(* PLC project EPEC_CU3.project, CODESYS V3.5 SP19 *)
(* stored: creationDateTime 2026-03-19T14:01:24.6293648+02:00, modificationDateTime 2026-03-19T14:01:24.6293648+02:00 *)

(* NOTE! NOTE! NOTE! NOTE! NOTE! NOTE! NOTE! NOTE! NOTE! NOTE! NOTE! This object is created by Epec MultiTool. User changes are overwritten when project is imported. Content: - EventCode channel IDs *)
{attribute 'qualified_only'}
{attribute 'strict'}
TYPE ChannelIDs : (Ch1 := 0, Ch2, Ch3, Ch4) BYTE;
END_TYPE

(* NOTE! NOTE! NOTE! NOTE! NOTE! NOTE! NOTE! NOTE! NOTE! NOTE! NOTE! This object is created by Epec MultiTool. User changes are overwritten when project is imported. Content: - EventCode device IDs *)
{attribute 'qualified_only'}
{attribute 'strict'}
TYPE DeviceIDs : (VoltageInput := 0, DigitalInput, CurrentInput, ParameterValidation) BYTE;
END_TYPE

TYPE IdentityObject : STRUCT
  VendorId : DWORD := 0;  (* Vendor ID *)
  ProductCode : DWORD := 0;  (* Product code *)
  Revision : DWORD := 0;  (* Revision number *)
  SerialNumber : DWORD := 0;  (* Serial number for control unit *)
END_STRUCT;
END_TYPE

{attribute 'qualified_only'}
{attribute 'location' := '16#800'}
{attribute 'strict'}
TYPE InitCanProtocolStates : (INIT_CANOPEN_PROTOCOLS := 1, INIT_CANOPEN_OD := 2, INIT_CANOPEN_PDO := 3, INIT_CANOPEN_OD_SAVE := 4, INIT_CANOPEN_OD_REORG := 5, INIT_J1939 := 6, INIT_PROTOCOLS_DONE := 7);
END_TYPE

TYPE IdentityObject : STRUCT
  VendorId : DWORD := 0;  (* Vendor ID *)
  ProductCode : DWORD := 0;  (* Product code *)
  Revision : DWORD := 0;  (* Revision number *)
  SerialNumber : DWORD := 0;  (* Serial number for control unit *)
END_STRUCT;
END_TYPE

VAR_GLOBAL CONSTANT  (* G_CONSTANTS - NOTE! NOTE! NOTE! NOTE! NOTE! NOTE! NOTE! NOTE! NOTE! NOTE! NOTE! This object is created by Epec MultiTool. User changes are overwritten when project is imported. Content: - Project specific constant definitions *)
  G_PARAMHANDLERKEYWORD : DWORD := 16#30C7E7D4;  (* Parameterhandler keyword *)
  G_PARAM_BLOCK_MAX_SIZE : WORD := WORD#1024;
  G_PARAMETER_SAVE_STATUS_ERROR : BYTE := BYTE#16#00;
  G_PARAMETER_SAVE_STATUS_DONE : BYTE := BYTE#16#01;
  G_PARAMETER_SAVE_STATUS_IN_PROGRESS : BYTE := BYTE#16#FF;
  G_SAFE_PARAMETERS_AUTHENTICATED : BYTE := BYTE#1;
  G_SAFE_PARAMETERS_NOT_AUTHENTICATED : BYTE := BYTE#0;
END_VAR

{attribute 'qualified_only'}
VAR_GLOBAL  (* G_CAN - NOTE! NOTE! NOTE! NOTE! NOTE! NOTE! NOTE! NOTE! NOTE! NOTE! NOTE! This object is created by Epec MultiTool. User changes are overwritten when project is imported. Content: - CAN definitions *)
  Channel1 : EPEC_CoreCANVXD.Channel;
END_VAR

{attribute 'qualified_only'}
{attribute 'location' := '16#800'}
VAR_GLOBAL  (* G_Common *)
  ParHandler : EPEC_PH.ParameterHandler;  (* Parameterhandler. Utility library for ODSave. Library handles parameter image modification. *)
  ParFileHandler : EPEC_PH.ParameterFileHandler;  (* ParameterFileHandler. Library handles parameter image saving to file and reading it. *)
  ParameterArea : ARRAY[1..EPEC_PH.Parameters.G_PARAMETER_FILE_SIZE] OF BYTE;  (* Parameter image *)
  ProjectKey : STRING(79) := 'KEeJGzzvbvqAy4c';  (* Project key, used for validating the response code *)
END_VAR


{attribute 'qualified_only'}
{attribute 'location' := '16#800'}
{attribute 'analysis' := '-6'}
VAR_GLOBAL  (* G_Logs *)
  ApplicationLog : EPEC_SERRLOG.ErrorLog;
  AppLogInitOK : BOOL;
END_VAR


{attribute 'qualified_only'}
{attribute 'location' := '16#800'}
VAR_GLOBAL  (* G_StatusFlags - NOTE! NOTE! NOTE! NOTE! NOTE! NOTE! NOTE! NOTE! NOTE! NOTE! NOTE! This object is created by Epec MultiTool. User changes are overwritten when project is imported. Content: - PLC_PRG status flags *)
  CANopenCan1NMTResetRequest : BOOL := FALSE;  (* Reset request flags tell if module is wanted to reset after current application cycle. *)
  CANopenCan2NMTResetRequest : BOOL := FALSE;
  CANopenCan3NMTResetRequest : BOOL := FALSE;
  CANopenCan4NMTResetRequest : BOOL := FALSE;
  CANopenCan5NMTResetRequest : BOOL := FALSE;
  CANopenCan6NMTResetRequest : BOOL := FALSE;
  CANopenCan7NMTResetRequest : BOOL := FALSE;
  CANopenCan8NMTResetRequest : BOOL := FALSE;
  CANopenCan9NMTResetRequest : BOOL := FALSE;
  CANopenCan10NMTResetRequest : BOOL := FALSE;
  CANopenCan11NMTResetRequest : BOOL := FALSE;
  CANopenCan12NMTResetRequest : BOOL := FALSE;
  CANopenCan13NMTResetRequest : BOOL := FALSE;
  CANopenCan14NMTResetRequest : BOOL := FALSE;
  CANopenCan15NMTResetRequest : BOOL := FALSE;
  CANopenCan16NMTResetRequest : BOOL := FALSE;
  CANopenCan17NMTResetRequest : BOOL := FALSE;
  CANopenCan18NMTResetRequest : BOOL := FALSE;
  CANopenCan19NMTResetRequest : BOOL := FALSE;
  CANopenCan20NMTResetRequest : BOOL := FALSE;
  CANopenCan21NMTResetRequest : BOOL := FALSE;
  CANopenCan22NMTResetRequest : BOOL := FALSE;
  CANopenCan23NMTResetRequest : BOOL := FALSE;
  CANopenCan24NMTResetRequest : BOOL := FALSE;
  CANopenCan25NMTResetRequest : BOOL := FALSE;
  CANopenCan26NMTResetRequest : BOOL := FALSE;
  CANopenCan27NMTResetRequest : BOOL := FALSE;
  CANopenCan28NMTResetRequest : BOOL := FALSE;
  CANopenCan29NMTResetRequest : BOOL := FALSE;
  CANopenCan30NMTResetRequest : BOOL := FALSE;
  CANopenCan31NMTResetRequest : BOOL := FALSE;
  CANopenCan32NMTResetRequest : BOOL := FALSE;
  CANopenCan33NMTResetRequest : BOOL := FALSE;
  CANopenCan34NMTResetRequest : BOOL := FALSE;
  CANopenCan35NMTResetRequest : BOOL := FALSE;
  CANopenCan36NMTResetRequest : BOOL := FALSE;
  CANopenCan37NMTResetRequest : BOOL := FALSE;
  CANopenCan38NMTResetRequest : BOOL := FALSE;
  CANopenCan39NMTResetRequest : BOOL := FALSE;
  CANopenCan40NMTResetRequest : BOOL := FALSE;
  CANopenCan41NMTResetRequest : BOOL := FALSE;
  CANopenCan42NMTResetRequest : BOOL := FALSE;
  CANopenCan43NMTResetRequest : BOOL := FALSE;
  CANopenCan44NMTResetRequest : BOOL := FALSE;
  CANopenCan45NMTResetRequest : BOOL := FALSE;
  CANopenCan46NMTResetRequest : BOOL := FALSE;
  CANopenCan47NMTResetRequest : BOOL := FALSE;
  CANopenCan48NMTResetRequest : BOOL := FALSE;
  CANopenCan49NMTResetRequest : BOOL := FALSE;
  CANopenCan50NMTResetRequest : BOOL := FALSE;
  CANopenCan51NMTResetRequest : BOOL := FALSE;
  CANopenCan52NMTResetRequest : BOOL := FALSE;
  CANopenCan53NMTResetRequest : BOOL := FALSE;
  CANopenCan54NMTResetRequest : BOOL := FALSE;
  CANopenCan55NMTResetRequest : BOOL := FALSE;
  CANopenCan56NMTResetRequest : BOOL := FALSE;
  CANopenCan57NMTResetRequest : BOOL := FALSE;
  CANopenCan58NMTResetRequest : BOOL := FALSE;
  CANopenCan59NMTResetRequest : BOOL := FALSE;
  CANopenCan60NMTResetRequest : BOOL := FALSE;
  CANopenCan61NMTResetRequest : BOOL := FALSE;
  CANopenCan62NMTResetRequest : BOOL := FALSE;
  CANopenCan63NMTResetRequest : BOOL := FALSE;
  CANopenCan64NMTResetRequest : BOOL := FALSE;
  CANopenCan65NMTResetRequest : BOOL := FALSE;
  CANopenCan66NMTResetRequest : BOOL := FALSE;
  CANopenCan67NMTResetRequest : BOOL := FALSE;
  CANopenCan68NMTResetRequest : BOOL := FALSE;
  CANopenCan69NMTResetRequest : BOOL := FALSE;
  CANopenCan70NMTResetRequest : BOOL := FALSE;
  CANopenCan71NMTResetRequest : BOOL := FALSE;
  CANopenCan72NMTResetRequest : BOOL := FALSE;
  CANopenCan73NMTResetRequest : BOOL := FALSE;
  CANopenCan74NMTResetRequest : BOOL := FALSE;
  CANopenCan75NMTResetRequest : BOOL := FALSE;
  CANopenCan76NMTResetRequest : BOOL := FALSE;
  CANopenCan77NMTResetRequest : BOOL := FALSE;
  CANopenCan78NMTResetRequest : BOOL := FALSE;
  CANopenCan79NMTResetRequest : BOOL := FALSE;
  CANopenCan80NMTResetRequest : BOOL := FALSE;
  CANopenCan81NMTResetRequest : BOOL := FALSE;
  CANopenCan82NMTResetRequest : BOOL := FALSE;
  CANopenCan83NMTResetRequest : BOOL := FALSE;
  CANopenCan84NMTResetRequest : BOOL := FALSE;
  CANopenCan85NMTResetRequest : BOOL := FALSE;
  CANopenCan86NMTResetRequest : BOOL := FALSE;
  CANopenCan87NMTResetRequest : BOOL := FALSE;
  CANopenCan88NMTResetRequest : BOOL := FALSE;
  CANopenCan89NMTResetRequest : BOOL := FALSE;
  CANopenCan90NMTResetRequest : BOOL := FALSE;
  CANopenCan91NMTResetRequest : BOOL := FALSE;
  CANopenCan92NMTResetRequest : BOOL := FALSE;
  CANopenCan93NMTResetRequest : BOOL := FALSE;
  CANopenCan94NMTResetRequest : BOOL := FALSE;
  CANopenCan95NMTResetRequest : BOOL := FALSE;
  CANopenCan96NMTResetRequest : BOOL := FALSE;
  CANopenCan97NMTResetRequest : BOOL := FALSE;
  CANopenCan98NMTResetRequest : BOOL := FALSE;
  CANopenCan99NMTResetRequest : BOOL := FALSE;
  CANopenCan100NMTResetRequest : BOOL := FALSE;
  CANopenCan101NMTResetRequest : BOOL := FALSE;
  CANopenCan102NMTResetRequest : BOOL := FALSE;
  CANopenCan103NMTResetRequest : BOOL := FALSE;
  CANopenCan104NMTResetRequest : BOOL := FALSE;
  CANopenCan105NMTResetRequest : BOOL := FALSE;
  SystemOk : BOOL := FALSE;
END_VAR

{attribute 'qualified_only'}
{attribute 'location' := '16#800'}
VAR_GLOBAL  (* G_SystemInfo - NOTE! NOTE! NOTE! NOTE! NOTE! NOTE! NOTE! NOTE! NOTE! NOTE! NOTE! This object is created by Epec MultiTool. User changes are overwritten when project is imported. Content: - System information common for all ODs. *)
  ProjectInfo : PROJECT_INFO;
  DeviceName : STRING(79);  (* 16#1008: Manufacturer device name *)
  HWVersion : STRING(79);  (* 16#1009: Manufacturer hardware version *)
  SWVersion : STRING(79);  (* 16#100A: Manufacturer software version *)
  Identity : IdentityObject;  (* 16#1018: Identity object *)
  ToolsVersion : ARRAY[1..1] OF DWORD;  (* 16#2030 Codesys version *)
  SoftwareInformation : ARRAY[1..10] OF STRING(79) := [''];  (* 16#2130 Software information Sub1: Application version Sub2: Additional version information Sub3: Reserved for future use Sub4: Reserved for future use Sub5: Reserved for future use Sub6: Reserved for future use Sub7: Reserved for future use Sub8: Reserved for future use Sub9: Reserved for future use Sub10: Reserved for future use *)
  MACAddress : ARRAY[1..6] OF BYTE := [6(0)];  (* 16#2140 MAC address Sub1: MAC address byte 1 Sub2: MAC address byte 2 Sub3: MAC address byte 3 Sub4: MAC address byte 4 Sub5: MAC address byte 5 Sub6: MAC address byte 6 *)
  EthernetConfiguration : ARRAY[1..50] OF BYTE := [50(0)];  (* 16#2141 Ethernet configuration Sub1: Ethernet enabled/disabled Sub2: DHCP on/off Sub3: Reserved Sub4: Reserved Sub5: Reserved Sub6: Reserved Sub7: Reserved Sub8: Reserved Sub9: Reserved Sub10: Reserved Sub11: Reserved Sub12: Reserved Sub13: Reserved Sub14: Reserved Sub15: Reserved Sub16: Reserved Sub17: Reserved Sub18: Netstatus Sub19: IP address highest byte Sub20: IP address 3rd byte Sub21: IP address 2nd byte Sub22: IP address lowest byte Sub23: Gateway highest byte Sub24: Gateway 3rd byte Sub25: Gateway 2nd byte Sub26: Gateway lowest byte Sub27: Netmask highest byte Sub28: Netmask 3rd byte Sub29: Netmask 2nd byte Sub30: Netmask first byte Sub31: Reserved Sub32: Reserved Sub33: Reserved Sub34: Reserved Sub35: Reserved Sub36: Reserved Sub37: Reserved Sub38: Reserved Sub39: Reserved Sub40: Reserved Sub41: Reserved Sub42: Reserved Sub43: Reserved Sub44: Reserved Sub45: Reserved Sub46: Reserved Sub47: Reserved Sub48: Reserved Sub49: Reserved Sub50: Reserved *)
END_VAR

{attribute 'qualified_only'}
{attribute 'global_init_slot' := '49991'}
VAR_GLOBAL  (* G_CANopen_CAN1 - NOTE! NOTE! NOTE! NOTE! NOTE! NOTE! NOTE! NOTE! NOTE! NOTE! NOTE! This object is created by Epec MultiTool User changes are overwritten when project is imported Content - CANopen protocol variable definitions *)
  Device : EPEC_CANopen.Device;  (* CAN device *)
  OD : EPEC_CANopen.OD;  (* Object Dictionary data *)
  ODEntrys : ARRAY[1..67] OF EPEC_CANopen.ODEntry;
  Protocols : ARRAY[1..5] OF EPEC_CANopen.ProtocolEntry;  (* Protocol data *)
  HBCallbacks : ARRAY[1..1] OF EPEC_CANopen.CANopenHBCallback := [(i_NodeID := 3, i_Time := G_CANopen_CAN1_VAR.HBCTimes[1], i_pNext := 0)];  (* Heartbeat producer/consumer *)
  HB : EPEC_CANopen.HBData;  (* Heartbeat producer/consumer protocol data *)
  HB_Handler : EPEC_CANopen.CANopenHB;  (* Heartbeat producer/consumer protocol handler *)
  MonitoredNodes : ARRAY[1..1] OF EPEC_CANopen.SlaveData := [(pHBCallback := ADR(HBCallbacks[1]), KeepAlive := FALSE, Reset := FALSE, Mandatory := TRUE, DisableStart := FALSE, QueryWithSDO := FALSE, ConfigurationDelay := 1000, SDOQueryInterval := 0, ConfigurationTimeout := 10)];  (* NMT *)
  NMT : EPEC_CANopen.NMTData;  (* NMT protocol data *)
  NMT_Handler : EPEC_CANopen.CANopenNMT;  (* NMT protocol handler *)
  SSDO : EPEC_CANopen.SSDOData;  (* SDO server protocol data *)
  SSDO_Handler : EPEC_CANopen.CANopenSDOServer;  (* SDO server protocol handler *)
  GFC : EPEC_CANopen.GFCData;  (* GFC protocol data *)
  GFC_Handler : EPEC_CANopen.CANopenGFC;  (* GFC protocol handler *)
  CSDOS : ARRAY[1..127] OF EPEC_CANopen.CANopenCSDO := [];  (* SDO client instances *)
  AppLogDomain : EPEC_CANopen.Domain;  (* 16#2171 Application log domain *)
  SaveAll : EPEC_ODSave.SaveODSaveAll;
  DeleteAll : EPEC_ODSave.SaveODDeleteAll;
  Initialize : EPEC_ODSave.SaveODInitialize;
  SaveData : ARRAY[0..3] OF EPEC_ODSave.SaveODSubIndexDescription := [(StartIndex := 16#1000, EndIndex := 16#FFFF, GroupNum := 1), (StartIndex := 16#1000, EndIndex := 16#1FFF, GroupNum := 1), (StartIndex := 16#2000, EndIndex := 16#FFFF, GroupNum := 1), (StartIndex := 16#0, EndIndex := 16#0, GroupNum := 1)];
  SaveSubData1010h : EPEC_ODSave.SaveODSubService;
  OD_ReOrg : EPEC_CANopen.CANopenODReOrg;
END_VAR

{attribute 'qualified_only'}
{attribute 'location' := '16#800'}
{attribute 'global_init_slot' := '49990'}
VAR_GLOBAL  (* G_CANopen_CAN1_VAR - NOTE! NOTE! NOTE! NOTE! NOTE! NOTE! NOTE! NOTE! NOTE! NOTE! NOTE! This object is created by Epec MultiTool User changes are overwritten when project is imported Content - *)
  OD_Error : EPEC_CANopen.Errors := EPEC_CANopen.Errors.NotInitialized;
  ODSave_Error : EPEC_ODSave.SaveODErrors;
  Callback_Error : EPEC_CANopen.Errors := EPEC_CANopen.Errors.NotInitialized;
  ProtocolAdded : ARRAY[1..5] OF BOOL := [5(0)];
  HBCTimes : ARRAY[1..1] OF UDINT := [UDINT#400];
  HB_Error : EPEC_CANopen.Errors := EPEC_CANopen.Errors.NotInitialized;
  NMT_Error : EPEC_CANopen.Errors := EPEC_CANopen.Errors.NotInitialized;
  SSDO_Error : EPEC_CANopen.Errors := EPEC_CANopen.Errors.NotInitialized;
  GFC_Error : EPEC_CANopen.Errors := EPEC_CANopen.Errors.NotInitialized;
  GFC_Status : BYTE;  (* GFC status *)
  CSDO_Error : EPEC_CANopen.Errors := EPEC_CANopen.Errors.NotInitialized;
  OD_REORG_Error : EPEC_CANopen.Errors := EPEC_CANopen.Errors.NotInitialized;
  OdReOrgReady : BOOL := FALSE;  (* OD Reorganize operation ready *)
  SaveSigns1010 : ARRAY[0..3] OF DWORD;
  InitProtocolsCanState : InitCanProtocolStates := InitCanProtocolStates.INIT_CANOPEN_PROTOCOLS;
END_VAR

{attribute 'qualified_only'}
{attribute 'location' := '16#800'}
{attribute 'analysis' := '-5, -6, -33, -43, -48'}
VAR_GLOBAL  (* G_CAN1_VAR - NOTE! NOTE! NOTE! NOTE! NOTE! NOTE! NOTE! NOTE! NOTE! NOTE! NOTE! This object is created by Epec MultiTool User changes are overwritten when project is imported Content - CANopen OD index data *)
  DeviceType_Device1 : UDINT := 405;  (* 16#1000 Information about the device type *)
  ErrorReg_Device1 : USINT := 0;  (* 16#1001 Error information *)
  TPDO_DUMMY : BYTE := 0;  (* 16#2128 PDO Dummy Variable Index *)
  RPDO_DUMMY : BYTE := 0;  (* 16#2129 PDO Dummy Variable Index *)
  Parameter_CSV_unique_ID : UINT := 16#0000;  (* 16#2131 Parameter CSV unique ID *)
END_VAR

(* This PRG contains non safety-related code. The following attribute is autogenerated. Do not remove. *)
{attribute 'location' := '16#800'}
PROGRAM NVMemory
  VAR_INPUT
    i_Initialize : BOOL := TRUE;
  END_VAR
  VAR_OUTPUT
    o_InitReady : BOOL;
  END_VAR

            IF i_Initialize THEN
	(*Init ParameterHandler to use Filesystem *)
	G_Common.ParFileHandler.Init(
		i_pParamHandler:= ADR(G_Common.ParHandler), 
		i_pParamArea:= ADR(G_Common.ParameterArea), 
		i_ParamAreaSize:= EPEC_PH.Parameters.G_PARAMETER_FILE_SIZE, 
		i_FileName:= 'parameters.img'); 

	IF G_Common.ParFileHandler.o_Ready THEN
		G_Common.ParHandler.Init(
			i_pParamArea:= ADR(G_Common.ParameterArea),
			i_ParamAreaSize:= EPEC_PH.Parameters.G_PARAMETER_FILE_SIZE,
			i_Keyword:= G_PARAMHANDLERKEYWORD,
			i_ParameterMaxDataSize:= G_PARAM_BLOCK_MAX_SIZE);

		o_InitReady:= TRUE;
	END_IF
ELSE

	G_Common.ParFileHandler.Update(i_Enable:=TRUE);


END_IF
            
          
END_PROGRAM

(* Tool version : '8.6.9547.24640' (MultiTool build version) Xml version : '1.0.0' (MultiTool xml file version) Control Unit : 'EPEC_CU3' (Name of the unit in MultiTool) Control Unit Type : 'CORE1-01-B' (Type of the unit in MultiTool, including the functional version) CODESYS Profile : 'CODESYS V3.5 SP19' (CODESYS profile that was selected in MultiTool) Device Description Version: '3.5.19.3' (Device description version that was selected in MultiTool) Export Time : '19.03.2026 14.01.24' (Date and time when exported from MultiTool) Export Path : 'C:\Codesys RPC\apps\CodesysRPC\EPEC_CU3' (Path where MultiTool exported) Project File : 'C:\Codesys RPC\apps\CodesysRPC\CodesysRPC.mtproject' (MultiTool project file name that was used) *)
{attribute 'location' := '16#800'}
PROGRAM PLC_PRG
  VAR_OUTPUT
    o_InitDone : BOOL := FALSE;
  END_VAR

            
// Initialize application log
IF NOT G_Logs.AppLogInitOK THEN
	G_Logs.AppLogInitOK := EPEC_SERRLOG.S_InitErrorLog(i_pErrorLog:= ADR(G_Logs.ApplicationLog));
END_IF

IF NOT o_InitDone AND G_Logs.AppLogInitOK THEN

    (* Code template non-safe FB initializations *)
    IF NOT Init_Entry.o_Ready THEN
        Init_Entry();
    ELSIF NOT Init_IO.o_Ready THEN
        Init_IO();
    ELSIF NOT NVMemory.o_InitReady THEN
        NVMemory(i_Initialize:=TRUE);
	ELSIF NOT Init_CAN.o_Ready THEN
		Init_CAN();
	ELSIF NOT Init_CANopen_CAN1.o_Ready THEN
		Init_CANopen_CAN1();

    ELSE
        (* User non-safe initialization *)
        MainInit(o_MainInitReady=>o_InitDone);
    END_IF
ELSE
    (* Non-safe actions to execute before non-safe main program *)
	G_CAN.Channel1.CheckMessages();
	Handle_CANopen_CAN1();


	Handle_Diagnostic();


    (* User non-safe main program *)
    Main();

    (* Non-safe actions to execute after non-safe main program *)

    NVMemory(i_Initialize:=FALSE);

    (* Boot application if NMT reset requested *)
    //IF G_StatusFlags.CANopenCan1NMTResetRequest OR G_StatusFlags.CANopenCan2NMTResetRequest THEN
    //    EPEC_SYSTEM.BOOT_APPLICATION_KILL_RTS();
    //END_IF
END_IF



              
          
END_PROGRAM

(* NOTE! NOTE! NOTE! NOTE! NOTE! NOTE! NOTE! NOTE! NOTE! NOTE! NOTE! This object is created by Epec MultiTool User changes are overwritten when project is imported Content - Initialization of CAN channels This PRG contains non safety-related code. The following attribute is autogenerated. Do not remove. *)
{attribute 'location' := '16#800'}
{attribute 'analysis' := '-9, -38'}
PROGRAM Init_CAN
  VAR_OUTPUT
    o_Ready : BOOL := FALSE;
    o_Error : BOOL := FALSE;
    o_CAN1InitError : EPEC_CANVXD.ERROR := EPEC_CANVXD.ERROR.CHANNEL_NOT_INITIALIZED;
  END_VAR

            G_CAN.Channel1.SetLoopback(i_LoopbackEnabled:=TRUE);
o_CAN1InitError := G_CAN.Channel1.InitCAN(i_Channel := 1, i_BitRate := EPEC_CANVXD.BITRATE_250K, i_Flags := 0);

IF EPEC_CANVXD.ERROR.NO_ERROR = o_CAN1InitError THEN
	o_Error := FALSE;
ELSE
	o_Error := TRUE;

	EPEC_SERRLOG.S_AddError_DWORD(i_ErrorCode:= ApplicationErrors.CAN_INIT, i_LibraryErrorCode:= INT_TO_DINT(o_CAN1InitError), i_Info1:= 0, i_Info2:= 1);
END_IF

o_Ready := TRUE;

          
END_PROGRAM

(* NOTE! NOTE! NOTE! NOTE! NOTE! NOTE! NOTE! NOTE! NOTE! NOTE! NOTE! This object is created by Epec MultiTool User changes are overwritten when project is imported Content - Set system information common for all ODs. This PRG contains non safety-related code. The following attribute is autogenerated. Do not remove. *)
{attribute 'location' := '16#800'}
{attribute 'analysis' := '-9, -19, -26'}
PROGRAM Init_Entry
  VAR_OUTPUT
    o_Ready : BOOL;
  END_VAR

            EPEC_HW.SystemParameters.ReadData();

/// 16#1008: Manufacturer device name
G_SystemInfo.DeviceName := EPEC_HW.SystemParameters.o_DeviceName;
 /// 16#1009: Manufacturer hardware version
G_SystemInfo.HWVersion := EPEC_HW.SystemParameters.o_HardwareVersion;
/// 16#100A: Manufacturer software version
G_SystemInfo.SWVersion := EPEC_HW.SystemParameters.o_SoftwareVersion;
/// 16#1018: Identity object 
G_SystemInfo.Identity.VendorId := EPEC_HW.SystemParameters.o_VendorId;          /// Vendor ID
G_SystemInfo.Identity.ProductCode := EPEC_HW.SystemParameters.o_ProductCode;    /// Product code
G_SystemInfo.Identity.Revision := EPEC_HW.SystemParameters.o_RevisionNumber;    /// Revision number
G_SystemInfo.Identity.SerialNumber := EPEC_HW.SystemParameters.o_SerialNumber;  /// Serial number for control unit
/// 16#2030 Codesys version
G_SystemInfo.ToolsVersion[1] := DWORD#50659328;

o_Ready:= TRUE;

          
END_PROGRAM

(* NOTE! NOTE! NOTE! NOTE! NOTE! NOTE! NOTE! NOTE! NOTE! NOTE! NOTE! This object is created by Epec MultiTool User changes are overwritten when project is imported Content - Non-safe system status update This PRG contains non safety-related code. The following attribute is autogenerated. Do not remove. *)
{attribute 'location' := '16#800'}
PROGRAM Handle_Diagnostic

            (* System Ok conditions *)
G_StatusFlags.SystemOk:=
		NOT Init_CAN.o_Error AND			(* No errors in bus init *)
		NOT Init_CANopen_CAN1.o_Error;



          
END_PROGRAM

(* NOTE! NOTE! NOTE! NOTE! NOTE! NOTE! NOTE! NOTE! NOTE! NOTE! NOTE! This object is created by Epec MultiTool User changes are overwritten when project is imported Content - CANopen initialization - Includes Init_CANopen_OD1 - CANopen data update This PRG contains non safety-related code. The following attribute is autogenerated. Do not remove. *)
{attribute 'location' := '16#800'}
{attribute 'analysis' := '-9, -19, -130'}
PROGRAM Init_CANopen_CAN1
  VAR_OUTPUT
    o_Ready : BOOL := FALSE;
    o_Error : BOOL := FALSE;
  END_VAR
  VAR
    odReOrgReady : BOOL := FALSE;
  END_VAR

            CASE G_CANopen_CAN1_VAR.InitProtocolsCanState OF

InitCanProtocolStates.INIT_CANOPEN_PROTOCOLS:
	G_CANopen_CAN1.Device.itfCanChannel:=G_CAN.Channel1; (*Connect device to can channel*)
	G_CANopen_CAN1.Device.NodeID := BYTE#5;
	G_CANopen_CAN1.NMT.NmtState:=EPEC_CANopen.NMTState.BootUp; (* Set NMT status to BOOTUP *)

	(*Initialize OD's data structures*)
	G_CANopen_CAN1.OD.EntryCount:=SIZEOF(G_CANopen_CAN1.ODEntrys)/SIZEOF(G_CANopen_CAN1.ODEntrys[1]); (*Max entries of given OD(CANopenDeviceODEntrys array)*)
	G_CANopen_CAN1.OD.InOrder:=FALSE; (*OD isn't in order*)
	G_CANopen_CAN1.OD.NextFree:=0; (*OD does not have any entries yet*)
	G_CANopen_CAN1.OD.pODEntry:=ADR(G_CANopen_CAN1.ODEntrys); (*Pointer to OD array*)

	(*Define NMT protocol*)
	G_CANopen_CAN1.Protocols[1].Protocol:=EPEC_CANopen.ProtocolType.NMT;
	G_CANopen_CAN1.Protocols[1].pData:=ADR(G_CANopen_CAN1.NMT);
	G_CANopen_CAN1.Protocols[1].itfProtocol:=G_CANopen_CAN1.NMT_Handler;
	G_CANopen_CAN1.Protocols[1].pError:=ADR(G_CANopen_CAN1_VAR.NMT_Error);
	G_CANopen_CAN1_VAR.ProtocolAdded[1] := CANopenDeviceAddProtocol( (* Add to protocol stack *)
		i_pDevice:=ADR(G_CANopen_CAN1.Device),
		i_pProtocol:=ADR(G_CANopen_CAN1.Protocols[1]),
	);

	(*Initialize NMT protocol*)
	IF G_CANopen_CAN1_VAR.ProtocolAdded[1] THEN
		G_CANopen_CAN1.NMT_Handler.Init(
			i_pDevice := ADR(G_CANopen_CAN1.Device),
			i_ThisIsMaster := FALSE,
			i_StartInterval :=  1000,
			i_pMonitoredNodes := ADR(G_CANopen_CAN1.MonitoredNodes),
			i_NumberOfNodes := 1,
			i_SimultaneousSlaveConfiguration := FALSE,
			i_pOdReOrg := ADR(G_CANopen_CAN1.OD_ReOrg),
			o_Error => G_CANopen_CAN1_VAR.NMT_Error
		);
	ELSE
		G_CANopen_CAN1_VAR.NMT_Error := EPEC_CANopen.Errors.ProtocolDataMissing;
	END_IF

	(*Define OD protocol*)
	G_CANopen_CAN1.Protocols[2].Protocol:=EPEC_CANopen.ProtocolType.OD;
	G_CANopen_CAN1.Protocols[2].pData:=ADR(G_CANopen_CAN1.OD);
	G_CANopen_CAN1.Protocols[2].pError:=ADR(G_CANopen_CAN1_VAR.OD_Error);
	G_CANopen_CAN1_VAR.ProtocolAdded[2] := CANopenDeviceAddProtocol( (* Add to protocol stack *)
		i_pDevice:=ADR(G_CANopen_CAN1.Device),
		i_pProtocol:=ADR(G_CANopen_CAN1.Protocols[2]),
	);
	IF NOT G_CANopen_CAN1_VAR.ProtocolAdded[2] THEN
		G_CANopen_CAN1_VAR.OD_Error := EPEC_CANopen.Errors.ProtocolDataMissing;
	END_IF

	(*Define HB protocol
	- Uses NMT and OD protocol data, thus need to be defined after them.
	*)
	G_CANopen_CAN1.HB.HeartBeat.PT := T#200MS; (* HB producer time *)
	G_CANopen_CAN1.HB.pHBCTimes := ADR(G_CANopen_CAN1_VAR.HBCTimes); (* HB consumer times *)

	G_CANopen_CAN1.Protocols[3].Protocol:=EPEC_CANopen.ProtocolType.HB;
	G_CANopen_CAN1.Protocols[3].pData:=ADR(G_CANopen_CAN1.HB);
	G_CANopen_CAN1.Protocols[3].itfProtocol:=G_CANopen_CAN1.HB_Handler;
	G_CANopen_CAN1.Protocols[3].pError:=ADR(G_CANopen_CAN1_VAR.HB_Error);
	G_CANopen_CAN1_VAR.ProtocolAdded[3] := CANopenDeviceAddProtocol( (* Add to protocol stack *)
		i_pDevice:=ADR(G_CANopen_CAN1.Device),
		i_pProtocol:=ADR(G_CANopen_CAN1.Protocols[3]),
	);

	(* Initialize HB protocol *)
	IF G_CANopen_CAN1_VAR.ProtocolAdded[3] THEN

		(* Add monitored nodes *)
		G_CANopen_CAN1.HB_Handler.AddCallbackToList(
			i_pDevice := ADR(G_CANopen_CAN1.Device),
			i_pCallback:=ADR(G_CANopen_CAN1.HBCallbacks[1]),
			o_Error => G_CANopen_CAN1_VAR.HB_Error
		);
		IF G_CANopen_CAN1_VAR.HB_Error = EPEC_CANopen.Errors.NoError THEN
			G_CANopen_CAN1.HB_Handler.Init(
				i_pDevice := ADR(G_CANopen_CAN1.Device),
				o_Error => G_CANopen_CAN1_VAR.HB_Error
			);
		END_IF
	ELSE
		G_CANopen_CAN1_VAR.HB_Error := EPEC_CANopen.Errors.ProtocolDataMissing;
	END_IF

	(*Define SSDO protocol*)
	G_CANopen_CAN1.Protocols[4].Protocol:=EPEC_CANopen.ProtocolType.SSDO;
	G_CANopen_CAN1.Protocols[4].pData:=ADR(G_CANopen_CAN1.SSDO);
	G_CANopen_CAN1.Protocols[4].itfProtocol:=G_CANopen_CAN1.SSDO_Handler;
	G_CANopen_CAN1.Protocols[4].pError:=ADR(G_CANopen_CAN1_VAR.SSDO_Error);
	G_CANopen_CAN1_VAR.ProtocolAdded[4] := CANopenDeviceAddProtocol( (* Add to protocol stack *)
		i_pDevice:=ADR(G_CANopen_CAN1.Device),
		i_pProtocol:=ADR(G_CANopen_CAN1.Protocols[4])
	);
	IF G_CANopen_CAN1_VAR.ProtocolAdded[4] THEN
		G_CANopen_CAN1.SSDO_Handler.Init(
			i_pDevice := ADR(G_CANopen_CAN1.Device),
			o_Error => G_CANopen_CAN1_VAR.SSDO_Error
		);
	ELSE
		G_CANopen_CAN1_VAR.SSDO_Error := EPEC_CANopen.Errors.ProtocolDataMissing;
	END_IF

	(*Define GFC protocol*)
	G_CANopen_CAN1.Protocols[5].Protocol:=EPEC_CANopen.ProtocolType.GFC;
	G_CANopen_CAN1.Protocols[5].pData:=ADR(G_CANopen_CAN1.GFC);
	G_CANopen_CAN1.Protocols[5].itfProtocol:=G_CANopen_CAN1.GFC_Handler;
	G_CANopen_CAN1.Protocols[5].pError:=ADR(G_CANopen_CAN1_VAR.GFC_Error);
	G_CANopen_CAN1_VAR.ProtocolAdded[5] := CANopenDeviceAddProtocol(  (* Add to protocol stack *)
		i_pDevice:=ADR(G_CANopen_CAN1.Device),
		i_pProtocol:=ADR(G_CANopen_CAN1.Protocols[5])
	);
	IF G_CANopen_CAN1_VAR.ProtocolAdded[5] THEN
		G_CANopen_CAN1.GFC_Handler.Init(
			i_pDevice := ADR(G_CANopen_CAN1.Device),
			i_pStatus:=ADR(G_CANopen_CAN1_VAR.GFC_Status),
			o_Error => G_CANopen_CAN1_VAR.GFC_Error
		);
	ELSE
		G_CANopen_CAN1_VAR.GFC_Error := EPEC_CANopen.Errors.ProtocolDataMissing;
	END_IF

	(* Init CSDO instance array for bus *)
	EPEC_CANopen.CANopenSDOManager.Init(
		i_pDevice:=ADR(G_CANopen_CAN1.Device),
		i_pCSDOArrayStart:=ADR(G_CANopen_CAN1.CSDOS),
		i_CSDOArraySize:=SIZEOF(G_CANopen_CAN1.CSDOS)/SIZEOF(G_CANopen_CAN1.CSDOS[1]),
		o_Error=>G_CANopen_CAN1_VAR.CSDO_Error
	);

	G_CANopen_CAN1_VAR.InitProtocolsCanState := InitCanProtocolStates.INIT_CANOPEN_OD;

InitCanProtocolStates.INIT_CANOPEN_OD:

	(* Add index data to OD *)
	Init_CANopen_OD1(o_Ready=>); (* Must be done before initing PDOs and SRDOs. *)

	IF Init_CANopen_OD1.o_Ready THEN
		G_CANopen_CAN1_VAR.InitProtocolsCanState := InitCanProtocolStates.INIT_CANOPEN_OD_SAVE;
	END_IF


InitCanProtocolStates.INIT_CANOPEN_OD_SAVE:

	(*Initialize OD save*)
	G_CANopen_CAN1.SaveAll.Init(i_pParamHandler:=ADR(G_Common.ParHandler));
	G_CANopen_CAN1.DeleteAll.Init(i_pParamHandler:=ADR(G_Common.ParHandler));
	G_CANopen_CAN1.SaveSubData1010h.pSaveSigns := ADR(G_CANopen_CAN1_VAR.SaveSigns1010[0]);
	G_CANopen_CAN1.SaveSubData1010h.NumOfEntrys := 4;
	G_CANopen_CAN1.SaveSubData1010h.pSaveIndexData := ADR(G_CANopen_CAN1.SaveData[0]);
	G_CANopen_CAN1.SaveData[3].itfSaveAll := G_CANopen_CAN1.SaveAll;
	G_CANopen_CAN1.SaveData[3].itfDeleteAll := G_CANopen_CAN1.DeleteAll;
	G_CANopen_CAN1.OD.pAdditionalData := ADR(G_CANopen_CAN1.SaveSubData1010h);

	IF G_CANopen_CAN1_VAR.OD_Error = EPEC_CANopen.Errors.NoError THEN
		G_CANopen_CAN1.Initialize(i_pOD:=ADR(G_CANopen_CAN1.OD), i_pParamHandler:=ADR(G_Common.ParHandler), o_Error => G_CANopen_CAN1_VAR.ODSave_Error);
	END_IF

	G_CANopen_CAN1.OD_ReOrg.Init(i_pOD := ADR(G_CANopen_CAN1.OD), i_NumOfODIndexPerCycle := 50);
	G_CANopen_CAN1.OD_ReOrg.Start();

	G_CANopen_CAN1_VAR.InitProtocolsCanState := InitCanProtocolStates.INIT_CANOPEN_OD_REORG;

InitCanProtocolStates.INIT_CANOPEN_OD_REORG:

	G_CANopen_CAN1.OD_ReOrg.Update(o_Ready => odReOrgReady, o_Error => G_CANopen_CAN1_VAR.OD_REORG_Error);

	IF odReOrgReady THEN
		(* Check all protocol init status flags *)
		IF G_CANopen_CAN1_VAR.NMT_Error = EPEC_CANopen.Errors.NoError AND
			G_CANopen_CAN1_VAR.SSDO_Error = EPEC_CANopen.Errors.NoError AND
			G_CANopen_CAN1_VAR.OD_Error = EPEC_CANopen.Errors.NoError AND
			G_CANopen_CAN1_VAR.HB_Error = EPEC_CANopen.Errors.NoError AND
			G_CANopen_CAN1_VAR.CSDO_Error = EPEC_CANopen.Errors.NoError AND
			G_CANopen_CAN1_VAR.GFC_Error = EPEC_CANopen.Errors.NoError AND
			G_CANopen_CAN1_VAR.OD_REORG_Error = EPEC_CANopen.Errors.NoError
		THEN
			o_Error := FALSE; (* No errors in protocol inits *)
		ELSE
			o_Error := TRUE;

			EPEC_SERRLOG.S_AddError_DWORD(i_ErrorCode:= ApplicationErrors.CANOPEN_INIT_NMT, i_LibraryErrorCode:= INT_TO_DINT(G_CANopen_CAN1_VAR.NMT_Error), i_Info1:= 0, i_Info2:= 1);
			EPEC_SERRLOG.S_AddError_DWORD(i_ErrorCode:= ApplicationErrors.CANOPEN_INIT_SSDO, i_LibraryErrorCode:= INT_TO_DINT(G_CANopen_CAN1_VAR.SSDO_Error), i_Info1:= 0, i_Info2:= 1);
			EPEC_SERRLOG.S_AddError_DWORD(i_ErrorCode:= ApplicationErrors.CANOPEN_INIT_OD, i_LibraryErrorCode:= INT_TO_DINT(G_CANopen_CAN1_VAR.OD_Error), i_Info1:= 0, i_Info2:= 1);
			EPEC_SERRLOG.S_AddError_DWORD(i_ErrorCode:= ApplicationErrors.CANOPEN_INIT_HB, i_LibraryErrorCode:= INT_TO_DINT(G_CANopen_CAN1_VAR.HB_Error), i_Info1:= 0, i_Info2:= 1);
			EPEC_SERRLOG.S_AddError_DWORD(i_ErrorCode:= ApplicationErrors.CANOPEN_INIT_CSDO, i_LibraryErrorCode:= INT_TO_DINT(G_CANopen_CAN1_VAR.CSDO_Error), i_Info1:= 0, i_Info2:= 1);
			EPEC_SERRLOG.S_AddError_DWORD(i_ErrorCode:= ApplicationErrors.CANOPEN_INIT_GFC, i_LibraryErrorCode:= INT_TO_DINT(G_CANopen_CAN1_VAR.GFC_Error), i_Info1:= 0, i_Info2:= 1);
			EPEC_SERRLOG.S_AddError_DWORD(i_ErrorCode:= ApplicationErrors.CANOPEN_INIT_OD_REORG, i_LibraryErrorCode:= INT_TO_DINT(G_CANopen_CAN1_VAR.OD_REORG_Error), i_Info1:= 0, i_Info2:= 1);

		END_IF

		o_Ready:=TRUE;
		G_CANopen_CAN1_VAR.InitProtocolsCanState := InitCanProtocolStates.INIT_PROTOCOLS_DONE;
	END_IF
END_CASE

          
END_PROGRAM

(* NOTE! NOTE! NOTE! NOTE! NOTE! NOTE! NOTE! NOTE! NOTE! NOTE! NOTE! This object is created by Epec MultiTool User changes are overwritten when project is imported Content - CANopen object dictionary initialization This PRG contains non safety-related code. The following attribute is autogenerated. Do not remove. *)
{attribute 'location' := '16#800'}
{attribute 'analysis' := '-19'}
PROGRAM Init_CANopen_OD1
  VAR_OUTPUT
    o_Ready : BOOL := FALSE;
  END_VAR

            CASE G_CANopen_CAN1_VAR.InitProtocolsCanState OF

InitCanProtocolStates.INIT_CANOPEN_OD:

	(*16#0001..16#0009 Default types *)
	G_CANopen_CAN1_VAR.OD_Error := EPEC_CANopen.CANopenODAddDefautTypes(
		i_pOD:= ADR(G_CANopen_CAN1.OD)
	);

	(* 16#1000 Information about the device type *)
	IF G_CANopen_CAN1_VAR.OD_Error = EPEC_CANopen.Errors.NoError THEN
		G_CANopen_CAN1_VAR.OD_Error := CANopenODAddLine(
			i_pOD := ADR(G_CANopen_CAN1.OD),(*Address of Object dictionary where index will be added*)
			i_Index := G_CANOPEN_ODINDEX_DEVICE_TYPE,
			i_ObjectCode := EPEC_CANopen.ObjectCode.OD_VAR,(*Type of index*)
			i_NumOfSubids := USINT#0,(*Number of subindexes*)
			i_TypeSpec := EPEC_CANopen.DataType.Deftype_UNSIGNED32,(*Index datatype, either user defined or standard CiA 301*)
			i_ObjectAccess := G_CANOPEN_OD_ACCESS_NOWRITE OR G_CANOPEN_OD_ACCESS_SUB0NOWRITE,
			i_Sub0data := USINT#0,(*Value of subindex0 in array or (def)struct*)
			i_pIndexData := ADR(G_CAN1_VAR.DeviceType_Device1),
			i_itfSDOHandler := DWORD#0
		);
	END_IF

	(* 16#1001 Error information *)
	IF G_CANopen_CAN1_VAR.OD_Error = EPEC_CANopen.Errors.NoError THEN
		G_CANopen_CAN1_VAR.OD_Error := CANopenODAddLine(
			i_pOD := ADR(G_CANopen_CAN1.OD),(*Address of Object dictionary where index will be added*)
			i_Index := G_CANOPEN_ODINDEX_ERROR_REGISTER,
			i_ObjectCode := EPEC_CANopen.ObjectCode.OD_VAR,(*Type of index*)
			i_NumOfSubids := USINT#0,(*Number of subindexes*)
			i_TypeSpec := EPEC_CANopen.DataType.Deftype_UNSIGNED8,(*Index datatype, either user defined or standard CiA 301*)
			i_ObjectAccess := G_CANOPEN_OD_ACCESS_NOWRITE OR G_CANOPEN_OD_ACCESS_SUB0NOWRITE,
			i_Sub0data := USINT#0,(*Value of subindex0 in array or (def)struct*)
			i_pIndexData := ADR(G_CAN1_VAR.ErrorReg_Device1),
			i_itfSDOHandler := DWORD#0
		);
	END_IF

	(* 16#1008 Manufacturer device name *)
	IF G_CANopen_CAN1_VAR.OD_Error = EPEC_CANopen.Errors.NoError THEN
		G_CANopen_CAN1_VAR.OD_Error := CANopenODAddLine(
			i_pOD := ADR(G_CANopen_CAN1.OD),(*Address of Object dictionary where index will be added*)
			i_Index := G_CANOPEN_ODINDEX_MF_DEVICE_NAME,
			i_ObjectCode := EPEC_CANopen.ObjectCode.OD_VAR,(*Type of index*)
			i_NumOfSubids := USINT#0,(*Number of subindexes*)
			i_TypeSpec := EPEC_CANopen.DataType.Deftype_STRING,(*Index datatype, either user defined or standard CiA 301*)
			i_ObjectAccess := G_CANOPEN_OD_ACCESS_NOWRITE OR G_CANOPEN_OD_ACCESS_SUB0NOWRITE,
			i_Sub0data := USINT#0,(*Value of subindex0 in array or (def)struct*)
			i_pIndexData := ADR(G_SystemInfo.DeviceName),
			i_itfSDOHandler := DWORD#0
		);
	END_IF

	(* 16#100A Manufacturer software version *)
	IF G_CANopen_CAN1_VAR.OD_Error = EPEC_CANopen.Errors.NoError THEN
		G_CANopen_CAN1_VAR.OD_Error := CANopenODAddLine(
			i_pOD := ADR(G_CANopen_CAN1.OD),(*Address of Object dictionary where index will be added*)
			i_Index := G_CANOPEN_ODINDEX_MF_SW_VERSION,
			i_ObjectCode := EPEC_CANopen.ObjectCode.OD_VAR,(*Type of index*)
			i_NumOfSubids := USINT#0,(*Number of subindexes*)
			i_TypeSpec := EPEC_CANopen.DataType.Deftype_STRING,(*Index datatype, either user defined or standard CiA 301*)
			i_ObjectAccess := G_CANOPEN_OD_ACCESS_NOWRITE OR G_CANOPEN_OD_ACCESS_SUB0NOWRITE,
			i_Sub0data := USINT#0,(*Value of subindex0 in array or (def)struct*)
			i_pIndexData := ADR(G_SystemInfo.SWVersion),
			i_itfSDOHandler := DWORD#0
		);
	END_IF

	(* 16#1018   Vendor ID *)
	IF G_CANopen_CAN1_VAR.OD_Error = EPEC_CANopen.Errors.NoError THEN
		G_CANopen_CAN1_VAR.OD_Error := CANopenODAddLine(
			i_pOD := ADR(G_CANopen_CAN1.OD),(*Address of Object dictionary where index will be added*)
			i_Index := G_CANOPEN_ODINDEX_IDENTITY_OBJECT,
			i_ObjectCode := EPEC_CANopen.ObjectCode.OD_ARRAY, (*Type of index*)
			i_NumOfSubids := USINT#4,(*Number of subindexes*)
			i_TypeSpec := EPEC_CANopen.DataType.Deftype_UNSIGNED32,(*Index of 16-bit deftype*)
			i_ObjectAccess := G_CANOPEN_OD_ACCESS_NOWRITE OR G_CANOPEN_OD_ACCESS_SUB0NOWRITE,
			i_Sub0data := USINT#4,(*Value of subindex0 in array or (def)struct*)
			i_pIndexData := ADR(G_SystemInfo.Identity),
			i_itfSDOHandler := DWORD#0
		);
	END_IF
	(* 16#2030   CodesysVersion *)
	IF G_CANopen_CAN1_VAR.OD_Error = EPEC_CANopen.Errors.NoError THEN
		G_CANopen_CAN1_VAR.OD_Error := CANopenODAddLine(
			i_pOD := ADR(G_CANopen_CAN1.OD),(*Address of Object dictionary where index will be added*)
			i_Index := 16#2030,
			i_ObjectCode := EPEC_CANopen.ObjectCode.OD_ARRAY, (*Type of index*)
			i_NumOfSubids := USINT#1,(*Number of subindexes*)
			i_TypeSpec := EPEC_CANopen.DataType.Deftype_UNSIGNED32,(*Index of 16-bit deftype*)
			i_ObjectAccess := G_CANOPEN_OD_ACCESS_NOWRITE OR G_CANOPEN_OD_ACCESS_SUB0NOWRITE,
			i_Sub0data := USINT#1,(*Value of subindex0 in array or (def)struct*)
			i_pIndexData := ADR(G_SystemInfo.ToolsVersion),
			i_itfSDOHandler := DWORD#0
		);
	END_IF

	(* 16#2128 PDO Dummy Variable Index *)
	IF G_CANopen_CAN1_VAR.OD_Error = EPEC_CANopen.Errors.NoError THEN
		G_CANopen_CAN1_VAR.OD_Error := CANopenODAddLine(
			i_pOD := ADR(G_CANopen_CAN1.OD),(*Address of Object dictionary where index will be added*)
			i_Index := 16#2128,
			i_ObjectCode := EPEC_CANopen.ObjectCode.OD_VAR,(*Type of index*)
			i_NumOfSubids := USINT#0,(*Number of subindexes*)
			i_TypeSpec := EPEC_CANopen.DataType.Deftype_UNSIGNED8,(*Index datatype, either user defined or standard CiA 301*)
			i_ObjectAccess := G_CANOPEN_OD_ACCESS_READWRITE,
			i_Sub0data := USINT#0,(*Value of subindex0 in array or (def)struct*)
			i_pIndexData := ADR(G_CAN1_VAR.TPDO_DUMMY),
			i_itfSDOHandler := DWORD#0
		);
	END_IF

	(* 16#2129 PDO Dummy Variable Index *)
	IF G_CANopen_CAN1_VAR.OD_Error = EPEC_CANopen.Errors.NoError THEN
		G_CANopen_CAN1_VAR.OD_Error := CANopenODAddLine(
			i_pOD := ADR(G_CANopen_CAN1.OD),(*Address of Object dictionary where index will be added*)
			i_Index := 16#2129,
			i_ObjectCode := EPEC_CANopen.ObjectCode.OD_VAR,(*Type of index*)
			i_NumOfSubids := USINT#0,(*Number of subindexes*)
			i_TypeSpec := EPEC_CANopen.DataType.Deftype_UNSIGNED8,(*Index datatype, either user defined or standard CiA 301*)
			i_ObjectAccess := G_CANOPEN_OD_ACCESS_READWRITE,
			i_Sub0data := USINT#0,(*Value of subindex0 in array or (def)struct*)
			i_pIndexData := ADR(G_CAN1_VAR.RPDO_DUMMY),
			i_itfSDOHandler := DWORD#0
		);
	END_IF

	(* 16#2130   Application version *)
	IF G_CANopen_CAN1_VAR.OD_Error = EPEC_CANopen.Errors.NoError THEN
		G_CANopen_CAN1_VAR.OD_Error := CANopenODAddLine(
			i_pOD := ADR(G_CANopen_CAN1.OD),(*Address of Object dictionary where index will be added*)
			i_Index := 16#2130,
			i_ObjectCode := EPEC_CANopen.ObjectCode.OD_ARRAY, (*Type of index*)
			i_NumOfSubids := USINT#10,(*Number of subindexes*)
			i_TypeSpec := EPEC_CANopen.DataType.Deftype_STRING,(*Index of 16-bit deftype*)
			i_ObjectAccess := G_CANOPEN_OD_ACCESS_NOWRITE OR G_CANOPEN_OD_ACCESS_SUB0NOWRITE,
			i_Sub0data := USINT#10,(*Value of subindex0 in array or (def)struct*)
			i_pIndexData := ADR(G_SystemInfo.SoftwareInformation),
			i_itfSDOHandler := DWORD#0
		);
	END_IF

	(* 16#2140   MAC address byte 1 *)
	IF G_CANopen_CAN1_VAR.OD_Error = EPEC_CANopen.Errors.NoError THEN
		G_CANopen_CAN1_VAR.OD_Error := CANopenODAddLine(
			i_pOD := ADR(G_CANopen_CAN1.OD),(*Address of Object dictionary where index will be added*)
			i_Index := 16#2140,
			i_ObjectCode := EPEC_CANopen.ObjectCode.OD_ARRAY, (*Type of index*)
			i_NumOfSubids := USINT#6,(*Number of subindexes*)
			i_TypeSpec := EPEC_CANopen.DataType.Deftype_UNSIGNED8,(*Index of 16-bit deftype*)
			i_ObjectAccess := G_CANOPEN_OD_ACCESS_NOWRITE OR G_CANOPEN_OD_ACCESS_SUB0NOWRITE,
			i_Sub0data := USINT#6,(*Value of subindex0 in array or (def)struct*)
			i_pIndexData := ADR(G_SystemInfo.MACAddress),
			i_itfSDOHandler := DWORD#0
		);
	END_IF

	(* 16#2141   Ethernet enabled/disabled *)
	IF G_CANopen_CAN1_VAR.OD_Error = EPEC_CANopen.Errors.NoError THEN
		G_CANopen_CAN1_VAR.OD_Error := CANopenODAddLine(
			i_pOD := ADR(G_CANopen_CAN1.OD),(*Address of Object dictionary where index will be added*)
			i_Index := 16#2141,
			i_ObjectCode := EPEC_CANopen.ObjectCode.OD_ARRAY, (*Type of index*)
			i_NumOfSubids := USINT#50,(*Number of subindexes*)
			i_TypeSpec := EPEC_CANopen.DataType.Deftype_UNSIGNED8,(*Index of 16-bit deftype*)
			i_ObjectAccess := G_CANOPEN_OD_ACCESS_READWRITE OR G_CANOPEN_OD_ACCESS_SUB0NOWRITE,
			i_Sub0data := USINT#50,(*Value of subindex0 in array or (def)struct*)
			i_pIndexData := ADR(G_SystemInfo.EthernetConfiguration),
			i_itfSDOHandler := DWORD#0
		);
	END_IF

	(* 16#2131 Parameter CSV unique ID *)
	IF G_CANopen_CAN1_VAR.OD_Error = EPEC_CANopen.Errors.NoError THEN
		G_CANopen_CAN1_VAR.OD_Error := CANopenODAddLine(
			i_pOD := ADR(G_CANopen_CAN1.OD),(*Address of Object dictionary where index will be added*)
			i_Index := 16#2131,
			i_ObjectCode := EPEC_CANopen.ObjectCode.OD_VAR,(*Type of index*)
			i_NumOfSubids := USINT#0,(*Number of subindexes*)
			i_TypeSpec := EPEC_CANopen.DataType.Deftype_UNSIGNED16,(*Index datatype, either user defined or standard CiA 301*)
			i_ObjectAccess := G_CANOPEN_OD_ACCESS_NOWRITE OR G_CANOPEN_OD_ACCESS_SUB0NOWRITE,
			i_Sub0data := USINT#0,(*Value of subindex0 in array or (def)struct*)
			i_pIndexData := ADR(G_CAN1_VAR.Parameter_CSV_unique_ID),
			i_itfSDOHandler := DWORD#0
		);
	END_IF

	(*16#2170 Application log error count *)
	IF G_CANopen_CAN1_VAR.OD_Error = EPEC_CANopen.Errors.NoError THEN
		G_CANopen_CAN1_VAR.OD_Error := CANopenODAddLine(
			i_pOD:= ADR(G_CANopen_CAN1.OD), (*Address of Object dictionary where index will be added *)
			i_Index:= 16#2170,
			i_ObjectCode:= EPEC_CANopen.ObjectCode.OD_VAR, (*Type of index*)
			i_NumOfSubids:= USINT#0,(*Number of subindexes*)
			i_TypeSpec:= EPEC_CANopen.DataType.Deftype_UNSIGNED32,(*Index of 32 - bit deftype *)
			i_ObjectAccess:= G_CANOPEN_OD_ACCESS_NOWRITE OR G_CANOPEN_OD_ACCESS_SUB0NOWRITE,
			i_Sub0data := USINT#0,(*Value of subindex0 in array or (def)struct*)
			i_pIndexData:= ADR(G_Logs.ApplicationLog.count),
			i_itfSDOHandler:= DWORD#0
		);
	END_IF

	(*16#2171 Application log domain *)
		IF G_CANopen_CAN1_VAR.OD_Error = EPEC_CANopen.Errors.NoError THEN
		G_CANopen_CAN1.AppLogDomain.DataSize:= SIZEOF(G_Logs.ApplicationLog.loglines) * 8;
		G_CANopen_CAN1.AppLogDomain.pData:= ADR(G_Logs.ApplicationLog.loglines);

		G_CANopen_CAN1_VAR.OD_Error := CANopenODAddLine(
			i_pOD:= ADR(G_CANopen_CAN1.OD), (*Address of Object dictionary where index will be added *)
			i_Index:= 16#2171,
			i_ObjectCode:= EPEC_CANopen.ObjectCode.OD_DOMAIN, (*Type of index*)
			i_NumOfSubids:= USINT#0,(*Number of subindexes*)
			i_TypeSpec:= EPEC_CANopen.DataType.Deftype_Domain,(*Domain deftype *)
			i_ObjectAccess:= G_CANOPEN_OD_ACCESS_NOWRITE,
			i_Sub0data:= USINT#0,(*Value of subindex0 in array or (def)struct*)
			i_pIndexData:= ADR(G_CANopen_CAN1.AppLogDomain),
			i_itfSDOHandler:= DWORD#0
		);
	END_IF

	o_Ready := TRUE;
END_CASE

          
END_PROGRAM

(* NOTE! NOTE! NOTE! NOTE! NOTE! NOTE! NOTE! NOTE! NOTE! NOTE! NOTE! This object is created by Epec MultiTool User changes are overwritten when project is imported Content - CANopen data update This PRG contains non safety-related code. The following attribute is autogenerated. Do not remove. *)
{attribute 'location' := '16#800'}
{attribute 'analysis' := '-9, -169'}
PROGRAM Handle_CANopen_CAN1
  VAR_OUTPUT
    o_Error : BOOL := FALSE;
  END_VAR

            (* Update callback data *)
IF G_CAN.Channel1.GetLatestError() <> DWORD#0 THEN
	G_CANopen_CAN1_VAR.Callback_Error := EPEC_CANopen.Errors.CallbackError;
ELSE
	G_CANopen_CAN1_VAR.Callback_Error := EPEC_CANopen.Errors.NoError;
END_IF

(* Update protocol data *)
G_CANopen_CAN1.HB_Handler.Update(
	i_Enable := TRUE,
	o_Error => G_CANopen_CAN1_VAR.HB_Error
);
G_CANopen_CAN1.NMT_Handler.Update(
	i_Enable := TRUE,
	o_Error => G_CANopen_CAN1_VAR.NMT_Error
);
G_CANopen_CAN1.SSDO_Handler.Update(
	i_Enable := TRUE,
	o_Error => G_CANopen_CAN1_VAR.SSDO_Error
);
G_CANopen_CAN1.GFC_Handler.Update(
	i_Enable := TRUE,
	o_Error => G_CANopen_CAN1_VAR.GFC_Error
);

G_CANopen_CAN1.OD_ReOrg.Update(o_Ready => , o_Error => G_CANopen_CAN1_VAR.OD_REORG_Error);

IF G_CANopen_CAN1_VAR.HB_Error = EPEC_CANopen.Errors.NoError AND
	G_CANopen_CAN1_VAR.NMT_Error = EPEC_CANopen.Errors.NoError AND
	G_CANopen_CAN1_VAR.SSDO_Error = EPEC_CANopen.Errors.NoError AND
	G_CANopen_CAN1_VAR.GFC_Error = EPEC_CANopen.Errors.NoError AND
	G_CANopen_CAN1_VAR.OD_REORG_Error = EPEC_CANopen.Errors.NoError
THEN
	o_Error := FALSE;
ELSE
	o_Error := TRUE;

	EPEC_SERRLOG.S_AddError_DWORD(i_ErrorCode:= ApplicationErrors.CANOPEN_UPDATE_HB, i_LibraryErrorCode:= INT_TO_DINT(G_CANopen_CAN1_VAR.HB_Error), i_Info1:= 0, i_Info2:= 1);
	EPEC_SERRLOG.S_AddError_DWORD(i_ErrorCode:= ApplicationErrors.CANOPEN_UPDATE_NMT, i_LibraryErrorCode:= INT_TO_DINT(G_CANopen_CAN1_VAR.NMT_Error), i_Info1:= 0, i_Info2:= 1);
	EPEC_SERRLOG.S_AddError_DWORD(i_ErrorCode:= ApplicationErrors.CANOPEN_UPDATE_SSDO, i_LibraryErrorCode:= INT_TO_DINT(G_CANopen_CAN1_VAR.SSDO_Error), i_Info1:= 0, i_Info2:= 1);
	EPEC_SERRLOG.S_AddError_DWORD(i_ErrorCode:= ApplicationErrors.CANOPEN_UPDATE_GFC, i_LibraryErrorCode:= INT_TO_DINT(G_CANopen_CAN1_VAR.GFC_Error), i_Info1:= 0, i_Info2:= 1);
	EPEC_SERRLOG.S_AddError_DWORD(i_ErrorCode:= ApplicationErrors.CANOPEN_UPDATE_OD_REORG, i_LibraryErrorCode:= INT_TO_DINT(G_CANopen_CAN1_VAR.OD_REORG_Error), i_Info1:= 0, i_Info2:= 1);

END_IF


(*Check for NMT reset *)
IF G_CANopen_CAN1.NMT.StateChanged THEN
	IF G_CANopen_CAN1.NMT.LastNmtCommand = EPEC_CANopen.NMTCommand.Reset OR
		G_CANopen_CAN1.NMT.LastNmtCommand = EPEC_CANopen.NMTCommand.ResetCommunication
	THEN
		(* If there is an NMT reset command for the IEC application CANopen device,
		   This is only informative, application decides how to react to the command *)
		G_StatusFlags.CANopenCan1NMTResetRequest := TRUE;
	END_IF
END_IF


          
END_PROGRAM

(* NOTE! NOTE! NOTE! NOTE! NOTE! NOTE! NOTE! NOTE! NOTE! NOTE! NOTE! This object is created by Epec MultiTool User changes are overwritten when project is imported Content - Init IO. This PRG contains safety-related code. The following attribute is autogenerated. Do not remove. *)
{attribute 'analysis' := '-9, -12'}
PROGRAM Init_IO
  VAR_OUTPUT
    o_Ready : SAFEBOOL := FALSE;
  END_VAR

            o_Ready:=TRUE;

          
END_PROGRAM
